// TwinCAT 3 PLC project tc_project_app
// ProgramVersion: 3.1.4022.6
// libraries:
//   Tc2_EtherCAT, * (Beckhoff Automation GmbH)
//   Tc2_MC2, * (Beckhoff Automation GmbH)
//   Tc2_Standard, * (Beckhoff Automation GmbH)
//   Tc2_SUPS, * (Beckhoff Automation GmbH)
//   Tc2_System, * (Beckhoff Automation GmbH)
//   Tc2_Utilities, * (Beckhoff Automation GmbH)
//   Tc3_MC2_AdvancedHoming, * (Beckhoff Automation GmbH)
//   Tc3_Module, * (Beckhoff Automation GmbH)
//   TcUnit, * (www.tcunit.org)
//   VisuDialogs, * (System)
// project tree:
//   / GlobalTextList.TcGTLO, NC_Task_1_SAF.TcTTO, PlcTask.TcTTO (not stored), Visualization Manager.TcVMO (not stored)
//   GVLs/ GVL_APP.TcGVL
//   POUs/ FB_BarnDoors.TcPOU, FB_CalculateAngle.TcPOU, FB_CalculateGap.TcPOU, gapUpdate.TcPOU, MAIN.TcPOU
//   tc_mca_std_lib/DUTs/ E_AxisParameters.TcTLEO (not stored), E_EncoderTypeClass.TcDUT (not stored), E_HomeSwitchTypeClass.TcDUT (not stored), E_HomingRoutines.TcTLEO (not stored), E_MotionFunctions.TcDUT (not stored), E_MotorTypeClass.TcDUT (not stored), E_RestorePosition.TcDUT (not stored), ST_AxisConfig.TcDUT (not stored), ST_AxisControl.TcDUT (not stored), ST_AxisDescription.TcDUT (not stored), ST_AxisInputs.TcDUT (not stored), ST_AxisPersistent.TcDUT (not stored), ST_GearAxis.TcDUT (not stored), ST_AxisStatus.TcDUT (not stored), ST_AxisStruct.TcDUT (not stored)
//   tc_mca_std_lib/ Error_Log_Visu.TcVIS (not stored), languageSupport.TcTLO (not stored), MainVisu.TcVIS (not stored), visuTextLinks.TcTLO (not stored)
//   tc_mca_std_lib/GVLs/ GVL.TcGVL (not stored)
//   tc_mca_std_lib/POUs/ChangeConfig/ FB_ReadFloatParameter.TcPOU (not stored), FB_ReadParameterInNc_v1_00.TcPOU (not stored), FB_WriteFloatParameter.TcPOU (not stored), FB_WriteParameterInNc_v1_00.TcPOU (not stored)
//   tc_mca_std_lib/POUs/Motion/ FB_Axis.TcPOU (not stored)
//   tc_mca_std_lib/POUs/Motion/Homing/ FB_Homing.TcPOU (not stored), FB_ReadNcVelocities.TcPOU (not stored)
//   Test/app_tests/ tcUNIT_APP_RUN.TcPOU (not stored)
//   Test/common/ FB_tcUNIT_common.TcPOU (not stored), tcUNIT_GVL.TcGVL (not stored)
//   Test/standard_library_tests/ FB_Axis_TEST.TcPOU (not stored), tcUNIT_STD_LIB_RUN.TcPOU (not stored)
// real-time tasks:
//   TASK PlcTask: cycle T#10ms, priority 20, ADS port 351
// motion (NC):
//   TASK NC-Task 1 SAF: cycle T#2ms, priority 4, ADS port 501
//   TASK NC-Task 1 SVB: cycle T#10ms, priority 8, ADS port 511
//   AXIS Blade 1A (id 1)
//     Dynamic: AccelerationMaximum=500, DecelerationMaximum=500, Acceleration=100, Deceleration=100, Jerk=500, OverrideType=4
//     Velo: RefSearch=0.5, RefSync=0.1, SlowManual=1, FastManual=2, Maximum=100
//     PositionAreaControl: Range=0.05
//     TargetPosControl: Range=0.05, Time=0.5
//     OtherSettings: AllowMotionCmdToSlave=true, PulseDistancePos=1, PulseDistanceNeg=1
//     encoder EncType=5
//       EncPara: ScaleFactorNumerator=60, ScaleFactorDenominator=4096, Offset=245686.8164, Inverse=true, ReferenceSystem=1
//         FilterTime: TPos=0.02, TVelo=0.04
//         ActPosCorrection: Time=0.02
//         Inc: RefSoftSyncMask=#x0000ffff
//     drive DrvType=24
//       Analog: VeloReferenz=600, TorqueScale=1, ScaleFactorActTorque=0.1
//       TimeComp: TaskDelayCycles=1
//     controller CtrType=3
//       CtrPara: PriorControlFactor=1
//         PosDiffControl: Enable=false, Range=0.5, Time=0.5
//         PID: PosKp=10, PosTn=1, PosTv=1, PosTd=1, DeadBandPosition=0.1
//         Observer: BandWidth=20
//   AXIS Blade 1B (id 2)
//     Dynamic: AccelerationMaximum=500, DecelerationMaximum=500, Acceleration=384, Deceleration=384, Jerk=1602.78
//     Velo: RefSearch=1, RefSync=1, SlowManual=1, FastManual=2, Maximum=100
//     PositionAreaControl: Range=0.2
//     TargetPosControl: Range=0.2, Time=0.5
//     OtherSettings: AllowMotionCmdToSlave=true, PulseDistancePos=1, PulseDistanceNeg=1
//     encoder EncType=5
//       EncPara: ScaleFactorNumerator=60, ScaleFactorDenominator=4096, Offset=-245743.330078125, ReferenceSystem=1
//         Inc: RefSoftSyncMask=#x0000ffff
//     drive DrvType=24
//       DrvPara: Inverse=true
//         Analog: VeloReferenz=600, TorqueScale=10, ScaleFactorActTorque=0.1
//         TimeComp: TaskDelayCycles=1
//     controller CtrType=1
//       CtrPara: PriorControlFactor=1
//         PosDiffControl: Range=0.5, Time=0.5
//         PID: PosKp=10
//         Observer: BandWidth=20
//   AXIS Blade 2A (id 3)
//     OtherSettings: AllowMotionCmdToSlave=true
//     encoder EncType=4
//       EncPara: MaxCount=#x0000ffff
//         Inc: RefSoftSyncMask=#x0000ffff
//     drive DrvType=24
//       Analog: ScaleFactorActTorque=0.1
//       TimeComp: TaskDelayCycles=1
//     controller CtrType=1
//       CtrPara: PriorControlFactor=1
//         Observer: BandWidth=20
//   AXIS Blade 2B (id 4)
//     OtherSettings: AllowMotionCmdToSlave=true
//     encoder EncType=4
//       EncPara: MaxCount=#x0000ffff
//         Inc: RefSoftSyncMask=#x0000ffff
//     drive DrvType=24
//       Analog: ScaleFactorActTorque=0.1
//       TimeComp: TaskDelayCycles=1
//     controller CtrType=1
//       CtrPara: PriorControlFactor=1
//         Observer: BandWidth=20
//   AXIS Blade 3A (id 5)
//     OtherSettings: AllowMotionCmdToSlave=true
//     encoder EncType=4
//       EncPara: MaxCount=#x0000ffff
//         Inc: RefSoftSyncMask=#x0000ffff
//     drive DrvType=24
//       Analog: ScaleFactorActTorque=0.1
//       TimeComp: TaskDelayCycles=1
//     controller CtrType=1
//       CtrPara: PriorControlFactor=1
//         Observer: BandWidth=20
//   AXIS Blade 3B (id 6)
//     OtherSettings: AllowMotionCmdToSlave=true
//     encoder EncType=4
//       EncPara: MaxCount=#x0000ffff
//         Inc: RefSoftSyncMask=#x0000ffff
//     drive DrvType=24
//       Analog: ScaleFactorActTorque=0.1
//       TimeComp: TaskDelayCycles=1
//     controller CtrType=1
//       CtrPara: PriorControlFactor=1
//         Observer: BandWidth=20
//   AXIS Momentum Slits (id 7)
//     OtherSettings: AllowMotionCmdToSlave=true
//     encoder EncType=4
//       EncPara: MaxCount=#x0000ffff
//         Inc: RefSoftSyncMask=#x0000ffff
//     drive DrvType=24
//       Analog: ScaleFactorActTorque=0.1
//       TimeComp: TaskDelayCycles=1
//     controller CtrType=1
//       CtrPara: PriorControlFactor=1
//         Observer: BandWidth=20
//   AXIS Gap 1 (mm) (id 8)
//     PositionAreaControl: Enable=false
//     TargetPosControl: Enable=false
//     OtherSettings: AllowMotionCmdToSlave=true
//     encoder EncType=16
//       EncPara: ScaleFactorNumerator=1, ScaleFactorDenominator=10000, MaxCount=#x0000ffff, ReferenceSystem=1
//     drive DrvType=5
//       Analog: ScaleFactorActTorque=0.1
//       TimeComp: TaskDelayCycles=1
//     controller CtrType=1
//       CtrPara: PriorControlFactor=1
//         PosDiffControl: Enable=false
//         Observer: BandWidth=20
//   AXIS Gap 2 (mm) (id 9)
//     OtherSettings: AllowMotionCmdToSlave=true
//     encoder EncType=1
//     drive DrvType=5
//       Analog: ScaleFactorActTorque=0.1
//       TimeComp: TaskDelayCycles=1
//     controller CtrType=1
//       CtrPara: PriorControlFactor=1
//         Observer: BandWidth=20
//   AXIS Gap 3 (mm) (id 10)
//     OtherSettings: AllowMotionCmdToSlave=true
//     encoder EncType=1
//     drive DrvType=5
//       Analog: ScaleFactorActTorque=0.1
//       TimeComp: TaskDelayCycles=1
//     controller CtrType=1
//       CtrPara: PriorControlFactor=1
//         Observer: BandWidth=20
// I/O:
//   DEVICE Device 1 (EtherCAT), AmsNetId 5.63.196.154.2.1
//     Term 1 (EK1200) [EK1200-5000 EtherCAT Power supply (2A E-Bus)]
//       Term 2 (EL1808) [EL1808 8Ch. Dig. Input 24V, 3ms]
//       Term 3 (EL2808) [EL2808 8Ch. Dig. Output 24V, 0.5A]
//       Term 4 (EL3214) [EL3214 4Ch. Ana. Input PT100 (RTD)]
//       Term 5 (EL1008) [EL1008 8Ch. Dig. Input 24V, 3ms]
//       Term 6 (EL1008) [EL1008 8Ch. Dig. Input 24V, 3ms]
//       Term 7 (EL1018) [EL1018 8Ch. Dig. Input 24V, 10µs]
//       Term 8 (EL2809) [EL2809 16Ch. Dig. Output 24V, 0.5A]
//       Term 9 (EL2809) [EL2809 16Ch. Dig. Output 24V, 0.5A]
//       Term 10 (EL6070-0033) [EL6070-0033 1Ch. Licence key terminal, individual licences]
//       Term 11 (EL9505) [EL9505 Power supply terminal 5V]
//       Term 12 (EL1252-0050) [EL1252-0050 2Ch. Fast Dig. Input 5V, 1µs, DC Latch]
//       Term 13 (EK1110) [EK1110 EtherCAT extension]
//     Term 14 (EK1101) [EK1101 EtherCAT Coupler (2A E-Bus, ID switch)]
//       Term 15 (EL5101) [EL5101 1Ch. Inc. Encoder 5V]
//       Term 16 (EL5101) [EL5101 1Ch. Inc. Encoder 5V]
//       Term 17 (EL5101) [EL5101 1Ch. Inc. Encoder 5V]
//       Term 18 (EL5101) [EL5101 1Ch. Inc. Encoder 5V]
//       Term 19 (EL5101) [EL5101 1Ch. Inc. Encoder 5V]
//       Term 20 (EL5101) [EL5101 1Ch. Inc. Encoder 5V]
//       Term 21 (EL5101) [EL5101 1Ch. Inc. Encoder 5V]
//       Term 30 (EL9011) [EL9011 End Terminal]
//     Term 22 (EK1101) [EK1101 EtherCAT Coupler (2A E-Bus, ID switch)]
//       Term 23 (EL7047) [EL7047 1Ch. Stepper motor output stage (50V, 5A)]
//       Term 24 (EL7047) [EL7047 1Ch. Stepper motor output stage (50V, 5A)]
//       Term 25 (EL7047) [EL7047 1Ch. Stepper motor output stage (50V, 5A)]
//       Term 26 (EL7047) [EL7047 1Ch. Stepper motor output stage (50V, 5A)]
//       Term 27 (EL7047) [EL7047 1Ch. Stepper motor output stage (50V, 5A)]
//       Term 28 (EL7047) [EL7047 1Ch. Stepper motor output stage (50V, 5A)]
//       Term 29 (EL7047) [EL7047 1Ch. Stepper motor output stage (50V, 5A)]
//       Term 31 (EL9011) [EL9011 End Terminal]
// variable links:
//   tc_project_app Instance <-> Device 1 (EtherCAT)/Term 1 (EK1200)/Term 5 (EL1008)
//     PlcTask Inputs/GVL.astAxes[1].stInputs.bLimitFwd <-> Channel 1/Input
//     PlcTask Inputs/GVL.astAxes[3].stInputs.bLimitFwd <-> Channel 5/Input
//     PlcTask Inputs/GVL.astAxes[5].stInputs.bLimitFwd <-> Channel 2/Input
//     PlcTask Inputs/GVL.astAxes[2].stInputs.bLimitBwd <-> Channel 3/Input
//     PlcTask Inputs/GVL.astAxes[4].stInputs.bLimitBwd <-> Channel 7/Input
//     PlcTask Inputs/GVL.astAxes[6].stInputs.bLimitBwd <-> Channel 4/Input
//   tc_project_app Instance <-> Device 1 (EtherCAT)/Term 1 (EK1200)/Term 6 (EL1008)
//     PlcTask Inputs/GVL.astAxes[1].stInputs.bLimitBwd <-> Channel 1/Input
//     PlcTask Inputs/GVL.astAxes[3].stInputs.bLimitBwd <-> Channel 5/Input
//     PlcTask Inputs/GVL.astAxes[5].stInputs.bLimitBwd <-> Channel 2/Input
//     PlcTask Inputs/GVL.astAxes[2].stInputs.bLimitFwd <-> Channel 3/Input
//     PlcTask Inputs/GVL.astAxes[4].stInputs.bLimitFwd <-> Channel 7/Input
//     PlcTask Inputs/GVL.astAxes[6].stInputs.bLimitFwd <-> Channel 4/Input
//   tc_project_app Instance <-> Device 1 (EtherCAT)/Term 1 (EK1200)/Term 7 (EL1018)
//     PlcTask Inputs/GVL.astAxes[1].stInputs.bHomeSensor <-> Channel 1/Input
//     PlcTask Inputs/GVL.astAxes[2].stInputs.bHomeSensor <-> Channel 3/Input
//     PlcTask Inputs/GVL.astAxes[3].stInputs.bHomeSensor <-> Channel 5/Input
//     PlcTask Inputs/GVL.astAxes[4].stInputs.bHomeSensor <-> Channel 7/Input
//     PlcTask Inputs/GVL.astAxes[5].stInputs.bHomeSensor <-> Channel 2/Input
//     PlcTask Inputs/GVL.astAxes[6].stInputs.bHomeSensor <-> Channel 4/Input
//   tc_project_app Instance <-> Device 1 (EtherCAT)/Term 1 (EK1200)/Term 8 (EL2809)
//     PlcTask Outputs/MAIN.bSwPower[{1..16}] <-> Channel {1..16}/Output  (16 links)
//   tc_project_app Instance <-> Device 1 (EtherCAT)/Term 1 (EK1200)/Term 9 (EL2809)
//     PlcTask Outputs/MAIN.bSwPower[17] <-> Channel 1/Output
//     PlcTask Outputs/MAIN.bSwPower[18] <-> Channel 2/Output
//     PlcTask Outputs/MAIN.bSwPower[19] <-> Channel 3/Output
//   tc_project_app Instance <-> NC-Task 1 SAF/Axes/Blade 1A
//     PlcTask Inputs/GVL.astAxes[1].Axis.NcToPlc <-> Outputs/ToPlc
//     PlcTask Outputs/GVL.astAxes[1].Axis.PlcToNc <-> Inputs/FromPlc
//   tc_project_app Instance <-> NC-Task 1 SAF/Axes/Blade 1B
//     PlcTask Inputs/GVL.astAxes[2].Axis.NcToPlc <-> Outputs/ToPlc
//     PlcTask Outputs/GVL.astAxes[2].Axis.PlcToNc <-> Inputs/FromPlc
//   tc_project_app Instance <-> NC-Task 1 SAF/Axes/Blade 2A
//     PlcTask Inputs/GVL.astAxes[3].Axis.NcToPlc <-> Outputs/ToPlc
//     PlcTask Outputs/GVL.astAxes[3].Axis.PlcToNc <-> Inputs/FromPlc
//   tc_project_app Instance <-> NC-Task 1 SAF/Axes/Blade 2B
//     PlcTask Inputs/GVL.astAxes[4].Axis.NcToPlc <-> Outputs/ToPlc
//     PlcTask Outputs/GVL.astAxes[4].Axis.PlcToNc <-> Inputs/FromPlc
//   tc_project_app Instance <-> NC-Task 1 SAF/Axes/Blade 3A
//     PlcTask Inputs/GVL.astAxes[5].Axis.NcToPlc <-> Outputs/ToPlc
//     PlcTask Outputs/GVL.astAxes[5].Axis.PlcToNc <-> Inputs/FromPlc
//   tc_project_app Instance <-> NC-Task 1 SAF/Axes/Blade 3B
//     PlcTask Inputs/GVL.astAxes[6].Axis.NcToPlc <-> Outputs/ToPlc
//     PlcTask Outputs/GVL.astAxes[6].Axis.PlcToNc <-> Inputs/FromPlc
//   tc_project_app Instance <-> NC-Task 1 SAF/Axes/Gap 1 (mm)
//     NC_Task_1_SAF Outputs/gapUpdate.fbCalcGap1.iGapSize <-> Enc/Inputs/In/nDataIn1
//     PlcTask Inputs/GVL.astAxes[8].Axis.NcToPlc <-> Outputs/ToPlc
//     PlcTask Outputs/GVL.astAxes[8].Axis.PlcToNc <-> Inputs/FromPlc
//   tc_project_app Instance <-> NC-Task 1 SAF/Axes/Gap 2 (mm)
//     NC_Task_1_SAF Outputs/gapUpdate.fbCalcGap2.iGapSize <-> Enc/Inputs/In/nDataIn1
//     PlcTask Inputs/GVL.astAxes[9].Axis.NcToPlc <-> Outputs/ToPlc
//     PlcTask Outputs/GVL.astAxes[9].Axis.PlcToNc <-> Inputs/FromPlc
//   tc_project_app Instance <-> NC-Task 1 SAF/Axes/Gap 3 (mm)
//     NC_Task_1_SAF Outputs/gapUpdate.fbCalcGap3.iGapSize <-> Enc/Inputs/In/nDataIn1
//     PlcTask Inputs/GVL.astAxes[10].Axis.NcToPlc <-> Outputs/ToPlc
//     PlcTask Outputs/GVL.astAxes[10].Axis.PlcToNc <-> Inputs/FromPlc
//   tc_project_app Instance <-> NC-Task 1 SAF/Axes/Momentum Slits
//     PlcTask Inputs/GVL.astAxes[7].Axis.NcToPlc <-> Outputs/ToPlc
//     PlcTask Outputs/GVL.astAxes[7].Axis.PlcToNc <-> Inputs/FromPlc

CONFIGURATION tc_project_app
    RESOURCE PLC ON TwinCAT3
        TASK NC_Task_1_SAF(INTERVAL := T#2ms, PRIORITY := 4);
        PROGRAM gapUpdate WITH NC_Task_1_SAF : gapUpdate;
    END_RESOURCE
END_CONFIGURATION

// ---- GVLs/GVL_APP.TcGVL
{attribute 'qualified_only'}
VAR_GLOBAL

END_VAR

VAR_GLOBAL CONSTANT
    nAXIS_NUM :   UINT:=10;
END_VAR

// ---- POUs/gapUpdate.TcPOU
//{attribute 'TcCallAfterOutputUpdate' }
PROGRAM gapUpdate
VAR
    fbCalcGap1 : FB_CalculateGap;
    fbCalcGap2 : FB_CalculateGap;
    fbCalcGap3 : FB_CalculateGap;
    //FB Variables for Muon Gates
    //StateMachine: INT;
    //i : UINT;
    //fPositionToSet : LREAL;
    //toggleExecute : BOOL;
    //fCalculatedPosition AT %Q*: REAL;
    //fCalculatedInt AT %Q* : DINT;
    
    ENC_CONSTANT : LREAL := 10000;
END_VAR

fbCalcGap1.AngleBladeA := GVL.astAxes[1].stStatus.fActPosition;
fbCalcGap1.AngleBladeB := GVL.astAxes[2].stStatus.fActPosition;
fbCalcGap1.ENC_CONSTANT:= ENC_CONSTANT;
fbCalcGap1();

fbCalcGap2.AngleBladeA := GVL.astAxes[3].stStatus.fActPosition;
fbCalcGap2.AngleBladeB := GVL.astAxes[4].stStatus.fActPosition;
fbCalcGap2.ENC_CONSTANT:= ENC_CONSTANT;
fbCalcGap2();

fbCalcGap3.AngleBladeA := GVL.astAxes[5].stStatus.fActPosition;
fbCalcGap3.AngleBladeB := GVL.astAxes[6].stStatus.fActPosition;
fbCalcGap3.ENC_CONSTANT:= ENC_CONSTANT;
fbCalcGap3();
//fCalculatedPosition:= fbCalcGap1.GapSize;
//fCalculatedPosition:= fCalculatedPosition*10000;
//fCalculatedInt:=  REAL_TO_DINT(fCalculatedPosition);

END_PROGRAM

// ---- POUs/FB_CalculateGap.TcPOU
//This function is used to calculate the gap size between two 'barn door' type blades
FUNCTION_BLOCK FB_CalculateGap

VAR_INPUT

AngleBladeA : LREAL;
AngleBladeB : LREAL;
fBladeSize : LREAL:=62.94;
fClosedGap : LREAL:=2.00;
ENC_CONSTANT : LREAL;
END_VAR

VAR_OUTPUT

GapSize : LREAL;
iGapSize AT %Q* : DINT;

END_VAR

VAR



END_VAR

GapSize := fClosedGap + fBladeSize*(2-(COS(DEG_TO_RAD(AngleBladeA)) + COS(DEG_TO_RAD(AngleBladeB))));
iGapSize := REAL_TO_DINT(GapSize * ENC_CONSTANT);

END_FUNCTION_BLOCK

// ---- POUs/FB_BarnDoors.TcPOU
FUNCTION_BLOCK FB_BarnDoors
VAR_INPUT
    bladeA  : UINT;
    bladeB  : UINT;
    gap     : UINT;
    fClosedGap  : LREAL;
    fBladeSize  : LREAL;
    
END_VAR
VAR_OUTPUT
END_VAR
VAR
    iState: INT;
    fPositionToSet : LREAL;
    fCalculatedPosition : REAL;
    fCalculatedInt AT %Q* : DINT;
    fbCalcGap : FB_CalculateGap;
    fbCalcAngle : FB_CalculateAngle;
    
    timeout: TON;
END_VAR

timeout.PT:=T#2S; //2second timeout to attempt rehomes
timeout();

fbCalcAngle.BladeSize:=fBladeSize;
fbCalcAngle.ClosedGap:=fClosedGap;


//Check switches and enables (wouldn't cause crash)
IF GVL.astAxes[bladeA].stStatus.bBwEnabled AND GVL.astAxes[bladeB].stStatus.bFwEnabled THEN
    GVL.astAxes[gap].stInputs.bLimitFwd:= TRUE;
ELSE
    GVL.astAxes[gap].stInputs.bLimitFwd:= FALSE;
END_IF

IF GVL.astAxes[bladeA].stStatus.bFwEnabled AND GVL.astAxes[bladeB].stStatus.bBwEnabled THEN
    GVL.astAxes[gap].stInputs.bLimitBwd:= TRUE;
ELSE
    GVL.astAxes[gap].stInputs.bLimitBwd:= FALSE;
END_IF

IF GVL.astAxes[bladeA].stStatus.bEnabled AND GVL.astAxes[bladeB].stStatus.bEnabled THEN
    GVL.astAxes[gap].stControl.bEnable:= TRUE;
ELSE
    GVL.astAxes[gap].stControl.bEnable:= FALSE;
END_IF

fbCalcAngle(GapSize:=GVL.astAxes[gap].stConfig.fPosition);

CASE iState OF
0://Wait for blade axes enabled
    IF GVL.astAxes[bladeA].stStatus.bEnabled AND GVL.astAxes[bladeB].stStatus.bEnabled THEN
        iState:=1;
	END_IF

1:
    IF (NOT GVL.astAxes[bladeA].stStatus.bHomed) OR (NOT GVL.astAxes[bladeB].stStatus.bHomed) THEN
        GVL.astAxes[bladeA].stControl.eCommand:=E_MotionFunctions.eHome;
        GVL.astAxes[bladeA].stControl.bExecute:=TRUE;
        GVL.astAxes[bladeB].stControl.eCommand:=E_MotionFunctions.eHome;
        GVL.astAxes[bladeB].stControl.bExecute:=TRUE;
	END_IF
    iState:= 2;

2://Wait for all axes calibrated, if bladeA AND bladeB calibrated, can direct home gap to the correct value
    IF (GVL.astAxes[bladeA].stStatus.bHomed AND GVL.astAxes[bladeB].stStatus.bHomed) THEN
        fbCalcGap(AngleBladeA:=GVL.astAxes[bladeA].stStatus.fActPosition,AngleBladeB:=GVL.astAxes[bladeB].stStatus.fActPosition,fBladeSize:= fBladeSize, fClosedGap:=fClosedGap);
        GVL.astAxes[gap].stControl.eCommand:= E_MotionFunctions.eHome;
        GVL.astAxes[gap].stConfig.eHomeSeq:= E_HomingRoutines.eHomeDirect;
        GVL.astAxes[gap].stConfig.fHomePosition:= fbCalcGap.GapSize;
        GVL.astAxes[gap].stControl.bExecute:=TRUE;
        iState:=3;
        timeout.IN:=TRUE;
    END_IF
    
3://Wait for calibration complete
    //IF (GVL.astAxes[bladeA].stStatus.bHomed) AND (GVL.astAxes[bladeB].stStatus.bHomed) THEN
        //iState:=10;    
    IF (GVL.astAxes[gap].stStatus.bHomed) THEN
        iState:=10;
	END_IF
    IF timeout.Q THEN
        timeout.IN:=FALSE;
        iState:=0;
	END_IF
    
10://Everything calibrated, monitor for commands to gap axis
//MoveAbs command
IF GVL.astAxes[gap].stControl.eCommand = E_MotionFunctions.eMoveAbsolute AND GVL.astAxes[gap].stControl.bExecute AND GVL.astAxes[gap].stStatus.bEnabled THEN
    fbCalcAngle(GapSize:=GVL.astAxes[gap].stConfig.fPosition);
    GVL.astAxes[bladeA].stControl.eCommand := E_MotionFunctions.eMoveAbsolute;
    GVL.astAxes[bladeA].stConfig.fPosition := fbCalcAngle.AngleBladeB;
    GVL.astAxes[bladeA].stConfig.fVelocity:=GVL.astAxes[gap].stConfig.fVelocity;
    GVL.astAxes[bladeA].stControl.bExecute:=TRUE;
    GVL.astAxes[bladeB].stControl.eCommand := E_MotionFunctions.eMoveAbsolute;
    GVL.astAxes[bladeB].stConfig.fPosition := fbCalcAngle.AngleBladeA;
    GVL.astAxes[bladeB].stConfig.fVelocity:=GVL.astAxes[gap].stConfig.fVelocity;
    GVL.astAxes[bladeB].stControl.bExecute:=TRUE;
END_IF
//Stop command
IF GVL.astAxes[gap].stControl.bStop THEN
    GVL.astAxes[bladeA].stControl.bStop:=TRUE;
    GVL.astAxes[bladeB].stControl.bStop:=TRUE;
END_IF
//Velocity command
IF GVL.astAxes[gap].stControl.eCommand = E_MotionFunctions.eMoveVelocity AND GVL.astAxes[gap].stControl.bExecute AND GVL.astAxes[gap].stStatus.bEnabled THEN
    GVL.astAxes[bladeA].stControl.eCommand := E_MotionFunctions.eMoveVelocity;
    GVL.astAxes[bladeA].stConfig.fVelocity:= -GVL.astAxes[gap].stConfig.fVelocity;
    GVL.astAxes[bladeA].stControl.bExecute:=TRUE;
    GVL.astAxes[bladeB].stControl.eCommand := E_MotionFunctions.eMoveVelocity;
    GVL.astAxes[bladeB].stConfig.fVelocity:=GVL.astAxes[gap].stConfig.fVelocity;
    GVL.astAxes[bladeB].stControl.bExecute:=TRUE;
END_IF
//Relative command
IF GVL.astAxes[gap].stControl.eCommand = E_MotionFunctions.eMoveRelative AND GVL.astAxes[gap].stControl.bExecute AND GVL.astAxes[gap].stStatus.bEnabled THEN
    fbCalcAngle(GapSize:=GVL.astAxes[gap].stStatus.fActPosition + GVL.astAxes[gap].stConfig.fPosition);
    GVL.astAxes[bladeA].stControl.eCommand := E_MotionFunctions.eMoveAbsolute;
    GVL.astAxes[bladeA].stConfig.fPosition := fbCalcAngle.AngleBladeB;
    GVL.astAxes[bladeA].stConfig.fVelocity:=GVL.astAxes[gap].stConfig.fVelocity;
    GVL.astAxes[bladeA].stControl.bExecute:=TRUE;
    GVL.astAxes[bladeB].stControl.eCommand := E_MotionFunctions.eMoveAbsolute;
    GVL.astAxes[bladeB].stConfig.fPosition := fbCalcAngle.AngleBladeA;
    GVL.astAxes[bladeB].stConfig.fVelocity:=GVL.astAxes[gap].stConfig.fVelocity;
    GVL.astAxes[bladeB].stControl.bExecute:=TRUE;
END_IF

999: //ERROR STATE
    GVL.astAxes[gap].stControl.bEnable:= FALSE;
    //Wait for reset of axes and block moves.
    IF NOT(GVL.astAxes[bladeA].stStatus.bError AND GVL.astAxes[bladeB].stStatus.bError) THEN
        iState:=0;
	END_IF
    
END_CASE

IF GVL.astAxes[bladeA].stStatus.bError OR GVL.astAxes[bladeB].stStatus.bError OR GVL.astAxes[gap].stStatus.bError THEN
    iState:=999;
END_IF
IF NOT GVL.astAxes[bladeA].stStatus.bEnabled OR NOT GVL.astAxes[bladeB].stStatus.bEnabled THEN
    iState:=0;
END_IF

END_FUNCTION_BLOCK

// ---- POUs/FB_CalculateAngle.TcPOU
//This function is used to calculate the blade angle of each in a pair of blades, based on a symetric gap size
FUNCTION_BLOCK FB_CalculateAngle

VAR_INPUT
GapSize : LREAL;
BladeSize : LREAL;
ClosedGap : LREAL;

END_VAR

VAR_OUTPUT
AngleBladeA : LREAL;
AngleBladeB : LREAL;

END_VAR

VAR

//BLADESIZE : LREAL:=62.94;	
//CLOSEDGAP : LREAL:=2.00;

END_VAR

IF GapSize<ClosedGap THEN
    AngleBladeA:=0;
    AngleBladeB:=0;
ELSIF GapSize > (2*BladeSize+ClosedGap) THEN
    AngleBladeA:=90;
    AngleBladeB:=90;
ELSE
    AngleBladeA := RAD_TO_DEG(ACOS((BladeSize + (ClosedGap/2) - (GapSize/2))/BladeSize));
    AngleBladeB := RAD_TO_DEG(-ACOS((BladeSize + (ClosedGap/2) - (GapSize/2))/BladeSize));  
END_IF

END_FUNCTION_BLOCK

// ---- POUs/MAIN.TcPOU
PROGRAM MAIN
VAR
    sVersion: STRING := '1.0.0';
    afbAxes: ARRAY [1..GVL_APP.nAXIS_NUM] OF FB_Axis;
    hmiAxisSelection: INT := 1; //Not possible to use local hmi variables for array indexes


(******Outputs: Power for Limit switches and Home Sensors (every 4th output)********)
    bSwPower AT %Q*: ARRAY [1..19] OF BOOL;
    i : INT;

//Startup, Shutdown and UPS
    fbUPS: FB_S_UPS_CX51x0;
    eUpsMode: E_S_UPS_Mode := eSUPS_WrPersistData_Shutdown;
    eStartUp: (eColdStart, eReadAxisFeedbackType, eCheckReadDone, eExecuteRestore, eCheckRestore, eFinishRestore);
    bPositionRestoreDone: BOOL := FALSE;
    bRestoreExecute: BOOL := FALSE;
    bExecuteReadEncRefSys: BOOL := FALSE;
    nRetry: INT;
    iAxes : UINT; //index for for loops in Position recovery actions
    afbReadEncRefSys: ARRAY [1..GVL_APP.nAXIS_NUM] OF MC_ReadParameter;
    afbRestorePosition: ARRAY [1..GVL_APP.nAXIS_NUM] OF MC_SetPosition;
    fbGetDeviceIdentification: FB_GetDeviceIdentification;
      
    fbBarnDoor1 :   FB_BarnDoors;
    fbBarnDoor2 :   FB_BarnDoors;
    fbBarnDoor3 :   FB_BarnDoors;
    
    //BACKLASH
    fbBacklashAxis3 : MC_BacklashCompensation;
    fBacklashTestVal : LREAL := 1.41;
    bBacklash   : BOOL;
    
    
    
    //demo test routine data
    fTargetPositions : ARRAY [1..8] OF LREAL;
    BLADE1A : INT:= 1;
    BLADE1B : INT:= 2;
    BLADE2A : INT:= 3;
    BLADE2B : INT:= 4;
    BLADE3A : INT:= 5;
    BLADE3B : INT:= 6;
    GAP1    : INT:= 8;
    GAP2    : INT:= 9;
    GAP3    : INT:= 10;
    bRunDemo    : BOOL :=FALSE;
    iDemoState  : INT:= 0;
    delayTimer : TON;
   
    
    
END_VAR

VAR PERSISTENT
    bRestoreOnStartup : BOOL;
END_VAR

DEMO();

POSITION_RECOVERY();
PROG();
AXES();

ACTION AXES:
FOR GVL.iAxis:=1 TO GVL_APP.nAXIS_NUM DO
    aFbAxes[GVL.iAxis](stAxisStruct:=gvl.astAxes[GVL.iAxis]);
END_FOR
END_ACTION

ACTION CHECK_UPS:
fbUPS(eUpsMode := eUpsMode);

IF eGlobalSUpsState = eSUPS_PowerFailure THEN
    //first cycle of powerfailure
    //execute code that should only be done once with each powerfailure, i.e. increase powerfailure counter
    bRestoreOnStartup := TRUE;
    STORE_PERSISTENT();
    RETURN;
ELSIF eGlobalSUpsState <> eSUPS_PowerOK THEN
    //next cycles of powerfailure
    //skip regular code execution for the remaining cycles of the powerfailure/writing of persistent data/quick shutdown...
    RETURN;
END_IF
END_ACTION

ACTION DEMO:
//Demo routine
GVL.astAxes[GAP1].stStatus.bDone:= GVL.astAxes[BLADE1A].stStatus.bDone AND GVL.astAxes[BLADE1B].stStatus.bDone;
GVL.astAxes[GAP2].stStatus.bDone:= GVL.astAxes[BLADE2A].stStatus.bDone AND GVL.astAxes[BLADE2B].stStatus.bDone;
GVL.astAxes[GAP3].stStatus.bDone:= GVL.astAxes[BLADE3A].stStatus.bDone AND GVL.astAxes[BLADE3B].stStatus.bDone;

delayTimer.PT:=T#1S;
delayTimer();

IF NOT bRunDemo THEN
    delayTimer.IN:=TRUE;
END_IF

IF bRunDemo THEN
    CASE iDemoState OF
        0: 
            IF delayTimer.Q THEN
                GVL.astAxes[GAP1].stControl.eCommand:=E_MotionFunctions.eMoveAbsolute;
                GVL.astAxes[GAP1].stConfig.fPosition:= 20;
                GVL.astAxes[GAP1].stConfig.fVelocity:= 5;
                GVL.astAxes[GAP1].stControl.bExecute:= TRUE;
                iDemoState:=1;
                delayTimer.IN:=FALSE;
			END_IF            
        1:
            IF GVL.astAxes[GAP1].stStatus.bDone THEN
                iDemoState:=2;
                delayTimer.IN:= TRUE;            
			END_IF
        2:
            IF delayTimer.Q THEN
                GVL.astAxes[GAP1].stControl.eCommand:=E_MotionFunctions.eMoveAbsolute;
                GVL.astAxes[GAP1].stConfig.fPosition:= 5;
                GVL.astAxes[GAP1].stConfig.fVelocity:= 5;
                GVL.astAxes[GAP1].stControl.bExecute:= TRUE;
                iDemoState:=3;
                delayTimer.IN:= FALSE;
            END_IF
        3:
            //IF GVL.astAxes[iGap1].stStatus.bDone AND GVL.astAxes[1].stStatus.bDone AND GVL.astAxes[2].stStatus.bDone THEN
            IF GVL.astAxes[GAP1].stStatus.bDone THEN
                iDemoState:=4;
                delayTimer.IN:= TRUE; 
			END_IF
        4: 
            IF delayTimer.Q THEN
                GVL.astAxes[GAP2].stControl.eCommand:=E_MotionFunctions.eMoveAbsolute;
                GVL.astAxes[GAP2].stConfig.fPosition:= 20;
                GVL.astAxes[GAP2].stConfig.fVelocity:= 5;
                GVL.astAxes[GAP2].stControl.bExecute:= TRUE;
                iDemoState:=5;
                delayTimer.IN:=FALSE;
			END_IF            
        5:
            IF GVL.astAxes[GAP2].stStatus.bDone THEN
                iDemoState:=6;
                delayTimer.IN:= TRUE;            
			END_IF
        6:
            IF delayTimer.Q THEN
                GVL.astAxes[GAP2].stControl.eCommand:=E_MotionFunctions.eMoveAbsolute;
                GVL.astAxes[GAP2].stConfig.fPosition:= 5;
                GVL.astAxes[GAP2].stConfig.fVelocity:= 5;
                GVL.astAxes[GAP2].stControl.bExecute:= TRUE;
                iDemoState:=7;
                delayTimer.IN:= FALSE;
            END_IF
        7:
            //IF GVL.astAxes[iGap1].stStatus.bDone AND GVL.astAxes[1].stStatus.bDone AND GVL.astAxes[2].stStatus.bDone THEN
            IF GVL.astAxes[GAP2].stStatus.bDone THEN
                iDemoState:=8;
                delayTimer.IN:= TRUE; 
			END_IF
        8: 
            IF delayTimer.Q THEN
                GVL.astAxes[GAP3].stControl.eCommand:=E_MotionFunctions.eMoveAbsolute;
                GVL.astAxes[GAP3].stConfig.fPosition:= 20;
                GVL.astAxes[GAP3].stConfig.fVelocity:= 5;
                GVL.astAxes[GAP3].stControl.bExecute:= TRUE;
                iDemoState:=9;
                delayTimer.IN:=FALSE;
			END_IF            
        9:
            IF GVL.astAxes[GAP3].stStatus.bDone THEN
                iDemoState:=10;
                delayTimer.IN:= TRUE;            
			END_IF
        10:
            IF delayTimer.Q THEN
                GVL.astAxes[GAP3].stControl.eCommand:=E_MotionFunctions.eMoveAbsolute;
                GVL.astAxes[GAP3].stConfig.fPosition:= 5;
                GVL.astAxes[GAP3].stConfig.fVelocity:= 5;
                GVL.astAxes[GAP3].stControl.bExecute:= TRUE;
                iDemoState:=11;
                delayTimer.IN:= FALSE;
            END_IF
        11:
            IF GVL.astAxes[GAP3].stStatus.bDone THEN
                iDemoState:=12;
                delayTimer.IN:= TRUE; 
			END_IF
            
        12: //all together now
            IF delayTimer.Q THEN
                GVL.astAxes[GAP3].stControl.eCommand:=E_MotionFunctions.eMoveAbsolute;
                GVL.astAxes[GAP3].stConfig.fPosition:= 50;
                GVL.astAxes[GAP3].stConfig.fVelocity:= 5;
                GVL.astAxes[GAP3].stControl.bExecute:= TRUE;
                GVL.astAxes[GAP2].stControl.eCommand:=E_MotionFunctions.eMoveAbsolute;
                GVL.astAxes[GAP2].stConfig.fPosition:= 50;
                GVL.astAxes[GAP2].stConfig.fVelocity:= 5;
                GVL.astAxes[GAP2].stControl.bExecute:= TRUE;
                GVL.astAxes[GAP1].stControl.eCommand:=E_MotionFunctions.eMoveAbsolute;
                GVL.astAxes[GAP1].stConfig.fPosition:= 50;
                GVL.astAxes[GAP1].stConfig.fVelocity:= 5;
                GVL.astAxes[GAP1].stControl.bExecute:= TRUE;
                iDemoState:=13;
                delayTimer.IN:= FALSE;
            END_IF
        13:
            IF GVL.astAxes[GAP3].stStatus.bDone AND GVL.astAxes[GAP2].stStatus.bDone AND GVL.astAxes[GAP1].stStatus.bDone THEN
                iDemoState:=14;
                delayTimer.IN:= TRUE; 
			END_IF
        14: //all together now
            IF delayTimer.Q THEN
                GVL.astAxes[GAP3].stControl.eCommand:=E_MotionFunctions.eMoveAbsolute;
                GVL.astAxes[GAP3].stConfig.fPosition:= 40;
                GVL.astAxes[GAP3].stConfig.fVelocity:= 5;
                GVL.astAxes[GAP3].stControl.bExecute:= TRUE;
                GVL.astAxes[GAP2].stControl.eCommand:=E_MotionFunctions.eMoveAbsolute;
                GVL.astAxes[GAP2].stConfig.fPosition:= 30;
                GVL.astAxes[GAP2].stConfig.fVelocity:= 5;
                GVL.astAxes[GAP2].stControl.bExecute:= TRUE;
                GVL.astAxes[GAP1].stControl.eCommand:=E_MotionFunctions.eMoveAbsolute;
                GVL.astAxes[GAP1].stConfig.fPosition:= 20;
                GVL.astAxes[GAP1].stConfig.fVelocity:= 5;
                GVL.astAxes[GAP1].stControl.bExecute:= TRUE;
                iDemoState:=15;
                delayTimer.IN:= FALSE;
            END_IF
        15:
            IF GVL.astAxes[GAP3].stStatus.bDone AND GVL.astAxes[GAP2].stStatus.bDone AND GVL.astAxes[GAP1].stStatus.bDone THEN
                iDemoState:=16;
                delayTimer.IN:= TRUE; 
			END_IF
        16: //all together now
            IF delayTimer.Q THEN
                GVL.astAxes[GAP3].stControl.eCommand:=E_MotionFunctions.eMoveAbsolute;
                GVL.astAxes[GAP3].stConfig.fPosition:= 20;
                GVL.astAxes[GAP3].stConfig.fVelocity:= 5;
                GVL.astAxes[GAP3].stControl.bExecute:= TRUE;
                GVL.astAxes[GAP2].stControl.eCommand:=E_MotionFunctions.eMoveAbsolute;
                GVL.astAxes[GAP2].stConfig.fPosition:= 30;
                GVL.astAxes[GAP2].stConfig.fVelocity:= 5;
                GVL.astAxes[GAP2].stControl.bExecute:= TRUE;
                GVL.astAxes[GAP1].stControl.eCommand:=E_MotionFunctions.eMoveAbsolute;
                GVL.astAxes[GAP1].stConfig.fPosition:= 40;
                GVL.astAxes[GAP1].stConfig.fVelocity:= 5;
                GVL.astAxes[GAP1].stControl.bExecute:= TRUE;
                iDemoState:=17;
                delayTimer.IN:= FALSE;
            END_IF
        17:
            IF GVL.astAxes[GAP3].stStatus.bDone AND GVL.astAxes[GAP2].stStatus.bDone AND GVL.astAxes[GAP1].stStatus.bDone THEN
                iDemoState:=18;
                delayTimer.IN:= TRUE; 
			END_IF
        18: //all together now
            IF delayTimer.Q THEN
                GVL.astAxes[GAP3].stControl.eCommand:=E_MotionFunctions.eMoveAbsolute;
                GVL.astAxes[GAP3].stConfig.fPosition:= 15;
                GVL.astAxes[GAP3].stConfig.fVelocity:= 5;
                GVL.astAxes[GAP3].stControl.bExecute:= TRUE;
                GVL.astAxes[GAP2].stControl.eCommand:=E_MotionFunctions.eMoveAbsolute;
                GVL.astAxes[GAP2].stConfig.fPosition:= 15;
                GVL.astAxes[GAP2].stConfig.fVelocity:= 5;
                GVL.astAxes[GAP2].stControl.bExecute:= TRUE;
                GVL.astAxes[GAP1].stControl.eCommand:=E_MotionFunctions.eMoveAbsolute;
                GVL.astAxes[GAP1].stConfig.fPosition:= 15;
                GVL.astAxes[GAP1].stConfig.fVelocity:= 5;
                GVL.astAxes[GAP1].stControl.bExecute:= TRUE;
                iDemoState:=19;
                delayTimer.IN:= FALSE;
            END_IF
        19:
            IF GVL.astAxes[GAP3].stStatus.bDone AND GVL.astAxes[GAP2].stStatus.bDone AND GVL.astAxes[GAP1].stStatus.bDone THEN
                iDemoState:=0;
                delayTimer.IN:= TRUE; 
			END_IF
    END_CASE
END_IF
END_ACTION

METHOD enableAxis : BOOL
VAR_INPUT
    iAxis : UINT;
END_VAR
GVL.astAxes[iAxis].stConfig.fOverride:=100;
GVL.astAxes[iAxis].stControl.bEnable:= TRUE;
END_METHOD

ACTION POSITION_RECOVERY:
fbGetDeviceIdentification(bExecute := TRUE);
IF (fbGetDeviceIdentification.stDevIdent.strHardwareSerialNo <> '0') THEN
    CHECK_UPS();
    RESTORE_POSITIONS();
END_IF
END_ACTION

ACTION PROG:
(*MUON BARN DOORS*)
(*This application uses a set position functionblock to update
the gap size value of a virtual axis based on two real world barn door blades.
The gap size is limited by the geometry of the jaws defined by the closed gap size and the blade size*)

//All outputs powering limits turned on.
FOR i:=1 TO 19 DO
    bSwPower[i]:= TRUE;
END_FOR

//Select homing routine to use for each axis
GVL.astAxes[1].stConfig.eHomeSeq:=E_HomingRoutines.eHomeToEncPulse_viaFwdLimit;
GVL.astAxes[2].stConfig.eHomeSeq:=E_HomingRoutines.eHomeToEncPulse_viaBwdLimit;
GVL.astAxes[3].stConfig.eHomeSeq:=E_HomingRoutines.eHomeToEncPulse_viaFwdLimit;
GVL.astAxes[4].stConfig.eHomeSeq:=E_HomingRoutines.eHomeToEncPulse_viaBwdLimit;
GVL.astAxes[5].stConfig.eHomeSeq:=E_HomingRoutines.eHomeToEncPulse_viaFwdLimit;
GVL.astAxes[6].stConfig.eHomeSeq:=E_HomingRoutines.eHomeToEncPulse_viaBwdLimit;

//Set calibrated home position for each axis
GVL.astAxes[1].stConfig.fHomePosition:=-11.189; //was -10.09  (-8.7)
GVL.astAxes[2].stConfig.fHomePosition:=-2.495; //was 13.75 (12.2)
GVL.astAxes[3].stConfig.fHomePosition:=-3.83; //was -3.19 (-4.19) (-2.55
GVL.astAxes[4].stConfig.fHomePosition:=15.61; //was 14.26 (15.66)
GVL.astAxes[5].stConfig.fHomePosition:=-10.097; //was -9.8
GVL.astAxes[6].stConfig.fHomePosition:=8.55; //9.45 (9.43)

//Call function blocks with blade numbers and gap geometry.
fbBarnDoor1(bladeA:=1,bladeB:=2,gap:=8,fClosedGap:=1.10,fBladeSize:=64.4175); //New blade sizes taken from survey data with Tony Millington. BLADE SIZE WAS 62.94
fbBarnDoor2(bladeA:=3,bladeB:=4,gap:=9,fClosedGap:=1.45,fBladeSize:=64.4475);
fbBarnDoor3(bladeA:=5,bladeB:=6,gap:=10,fClosedGap:=1.49,fBladeSize:=64.4005);
END_ACTION

ACTION RESTORE_POSITIONS:
//This ACT will restore the position of an incremental axis on startup with the act position it read before losing power.
//It checks the type of axis, 0=incremental, and that the axis was stationary at shut down.
//Because 0 equates to incremental we also need to check that the data is valid, otherwise by default it would restore all axes.
//By default an axis will not restore the position unless it is set to opt-in, i.e. GVL.aAxes[iAxes].stConfig.eRestorePosition is non-zero.
//This needs to be initialised somewhere in TwinCAT code otherwise it will not be available at start up.
//A restore will only be performed on a loss of power, this code shouldn't make any changes on a reset cold, a rest origin or a download.
//There is a enum to allow for different types of restore modes, currently only one is implemented.
//0 'DontRestore'
//1 'RestoreWithoutHome' -restores the position using a set position fb and does not set the home bit in the axis struct.
//Note from Beckhoff: "A maximum of 1 MB persistent data can be reliably saved over the entire service life."

IF bRestoreOnStartup AND eGlobalSUpsState = eSUPS_PowerOK THEN
    bRestoreOnStartup := FALSE;
    bRestoreExecute := TRUE;
END_IF

//Upon startup bPositionRestoreDone will be set to FALSE, after successfully completing the following code it will be set TRUE
//and should stay TRUE for the rest of the time the PLC is operational, thus this routine should only be completed once.
IF bRestoreExecute AND NOT bPositionRestoreDone THEN
    //Cycle through function blocks that read the encoder reference system i.e. whether axis is incremental or absolute
    //Result stored in Value, 0=Inc 1=Abs, execute set during the case statement
    FOR iAxes := 1 TO GVL_APP.nAXIS_NUM DO
        afbReadEncRefSys[iAxes](
          Axis := GVL.astAxes[iAxes].Axis,
          Enable := bExecuteReadEncRefSys,
          ParameterNumber := MC_AxisParameter.AxisEncoderReferenceSystem,
          ReadMode := E_READMODE.READMODE_ONCE);
    END_FOR

    //Cycle through set position function blocks for each axis
    FOR iAxes := 1 TO GVL_APP.nAXIS_NUM DO
        afbRestorePosition[iAxes](
         Axis := GVL.astAxes[iAxes].Axis,
         Position := astAxesPersistent[iAxes].fPositionAtShutdown);
    END_FOR

    CASE eStartUp OF
        eColdStart:
        //First cycle of the PLC, do nothing just give one cycle for variables to initialise
            IF NOT bPositionRestoreDone THEN
                eStartUp := eReadAxisFeedbackType;
                nRetry := 0;
            END_IF

        eReadAxisFeedbackType:
        //Exectute the function blocks to read the encoder reference system (0=inc OR 1=ABS)
            bExecuteReadEncRefSys := TRUE;
            eStartUp := eCheckReadDone;

        eCheckReadDone:
        //Check the encoder reference system has been read for all axis -> if busy then continue with PLC cycle and check again next time.
        //If afbReadEncRefSys not started then go back a step.
        //If any axes result in an error the code will get stuck here, this happens if GVL_APP.nAXIS_NUM is not set correctly
            FOR iAxes := 1 TO GVL_APP.nAXIS_NUM DO
                IF afbReadEncRefSys[iAxes].Valid = FALSE THEN
                    IF afbReadEncRefSys[iAxes].Busy = TRUE THEN
                        //Exit MAIN.STARTUP Action and wait till next cycle, needs to cycle through whole program in order for data to update
                        RETURN;
                    ELSE
                        //Sometimes the code gets here and the afbReadEncRefSys[iAxes] misses the rising edge. If  the code gets here it means
                        //valid=FALSE and .busy=FALSE which indicateds the FB probably hasn't started and thus needs to see a rising edge.
                        //Set execute to low, Exit MAIN.STARTUP and go back a step in the CASE statement.
                        bExecuteReadEncRefSys := FALSE;
                        eStartUp := eReadAxisFeedbackType;
                        nRetry := nRetry + 1; //counter used for troubleshooting to see how many cycles it takes before afbReadEncRefSys function blocks are read correctly
                        RETURN;
                    END_IF
                END_IF
            END_FOR
            //If the code gets here all axes either have .valid=TRUE for all axes
            eStartUp := eExecuteRestore;

        eExecuteRestore:
        //Execute position restore by setting afbRestorePosition.execute = TRUE
            FOR iAxes := 1 TO GVL_APP.nAXIS_NUM DO
                IF afbReadEncRefSys[iAxes].Valid = TRUE AND afbReadEncRefSys[iAxes].Value = 0 AND NOT(astAxesPersistent[iAxes].bMovingAtShutdown) THEN
                    IF GVL.astAxes[iAxes].stConfig.eRestorePosition = E_RestorePosition.eRestoreWithoutHome THEN
                        afbRestorePosition[iAxes].Execute := TRUE;
                    END_IF
                END_IF
            END_FOR
            eStartUp := eCheckRestore;

        eCheckRestore:
        //Check the set position fbs are finished
        //Nothing actually happens if the restore is not done, the code just returns from here each cycle and the
        //bPositionRestoreDone will never get set to TRUE and will take up cycle time
            FOR iAxes := 1 TO GVL_APP.nAXIS_NUM DO
                IF afbReadEncRefSys[iAxes].Valid = TRUE AND afbReadEncRefSys[iAxes].Value = 0 AND NOT(astAxesPersistent[iAxes].bMovingAtShutdown) THEN
                    IF GVL.astAxes[iAxes].stConfig.eRestorePosition = E_RestorePosition.eRestoreWithoutHome THEN
                        IF NOT afbRestorePosition[iAxes].Done THEN
                            RETURN;
                        END_IF
                    END_IF
                END_IF
            END_FOR
            eStartUp := eFinishRestore;

        eFinishRestore:
        //Remove execute = TRUE for afbRestorePosition
            FOR iAxes := 1 TO GVL_APP.nAXIS_NUM DO
                afbRestorePosition[iAxes].Execute := FALSE;
            END_FOR
            bPositionRestoreDone := TRUE;
            bRestoreExecute := FALSE;
    END_CASE
END_IF
END_ACTION

ACTION STORE_PERSISTENT:
FOR iAxes := 1 TO GVL_APP.nAXIS_NUM DO
    astAxesPersistent[iAxes].fPositionAtShutdown := GVL.astAxes[iAxes].Axis.NcToPlc.ActPos;
    IF GVL.astAxes[iAxes].Axis.NcToPlc.ActVelo <> 0 THEN
        astAxesPersistent[iAxes].bMovingAtShutdown := TRUE;
    ELSE
        astAxesPersistent[iAxes].bMovingAtShutdown := FALSE;
    END_IF
    astAxesPersistent[iAxes].bMovingAtShutdown := astAxesPersistent[iAxes].bMovingAtShutdown OR GVL.astAxes[iAxes].Axis.Status.Moving;
END_FOR
END_ACTION

END_PROGRAM

// ---- GlobalTextList.TcGTLO
TEXTLIST GlobalTextList
  951 = '%2.2f'
  317 = '%2.3f'
  543 = '%2.4f'
  878 = '%d'
  706 = '%i'
  940 = '%x'
  703 = 'Acknowledge'
  710 = 'Active:'
  952 = 'actPos'
  953 = 'actVel'
  110 = 'AXESMAX'
  107 = 'axisSel'
  945 = 'bBusy'
  950 = 'bBwEnabled'
  946 = 'bDone'
  943 = 'bEnabled'
  941 = 'bError'
  102 = 'bExecute'
  949 = 'bFwEnabled'
  297 = 'bGeared'
  948 = 'bHomed'
  947 = 'bResetDone'
  944 = 'bWarning'
  704 = 'Clear All'
  986 = 'ehomeDirect'
  198 = 'eHomeToEncPulse_Bwd'
  510 = 'eHomeToEncPulse_Fwd'
  287 = 'eHomeToEncPulse_viaBwdLimit'
  683 = 'eHomeToEncPulse_viaFwdLimit'
  312 = 'eHomeToLimit_Bwd'
  635 = 'eHomeToLimit_Fwd'
  150 = 'eHomeToRef_Bwd'
  861 = 'eHomeToRef_Fwd'
  104 = 'ENABLE'
  106 = 'ENABLE BW'
  105 = 'ENABLE FW'
  109 = 'English'
  939 = 'errID'
  701 = 'Error #'
  705 = 'Error #:'
  702 = 'Error Log'
  707 = 'Errors:'
  768 = 'eWriteParameter'
  955 = 'fAcceleration'
  956 = 'fDeceleration'
  531 = 'fHomeFinishDistance'
  613 = 'fHomePosition'
  957 = 'fPosition'
  149 = 'fRatio'
  781 = 'fReadAxisParameter'
  708 = 'Free Entries:'
  954 = 'fVelocity'
  688 = 'fWriteAxisParameter'
  299 = 'gearIn'
  717 = 'gearInMultiMaster'
  300 = 'gearOut'
  718 = 'HOME'
  711 = 'Inactive:'
  116 = 'jogBw'
  117 = 'jogFw'
  298 = 'masterGear'
  111 = 'moveAbsolute'
  114 = 'moveModulo'
  113 = 'moveRelative'
  112 = 'moveVelocity'
  575 = 'nIndex'
  709 = 'Overflows:'
  942 = 'reset'
  115 = 'stop'
  108 = 'Test Language'
  103 = 'toggle'
END_TEXTLIST
